// Mitsubishi GX Works2 project: m08   PLC: Q02/Q02H

PROGRAM MAIN
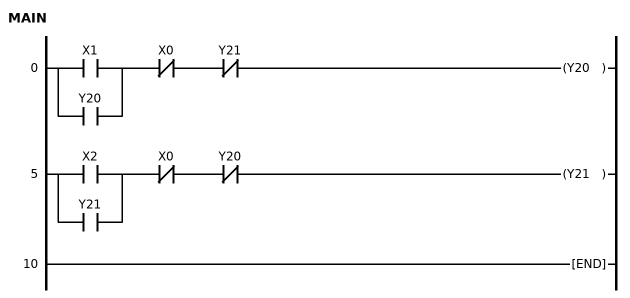
0     LD      X1
      OR      Y20
      ANI     X0
      ANI     Y21
      OUT     Y20
5     LD      X2
      OR      Y21
      ANI     X0
      ANI     Y20
      OUT     Y21
10    END
END_PROGRAM
